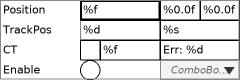
VISUALIZATION _VISU_WorkerDefGrid  // 240x80
VAR_IN_OUT
	m_Inst : FB_WorkerDefGrid;
END_VAR
    Rectangle (0,0 240x60)
    Rectangle (80,20 80x20), "%d", text variable: m_Inst._nTrackOffset
    Rectangle (0,0 80x20), "Position"
    Rectangle (0,20 80x20), "TrackPos"
    Rectangle (80,0 80x20), "%f", text variable: m_Inst.fPosition
        OnMouseClick: write the text variable via Default
    Rectangle (160,20 80x20), "%s", text variable: m_Inst._nTrackPosDomain
    Rectangle (160,0 40x20), "%0.0f", text variable: m_Inst._fPrintResolution
    Rectangle (200,0 40x20), "%0.0f", text variable: m_Inst._fSubPxResolution
    Rectangle (0,40 80x20), "CT"
    RoundedRectangle (80,40 20x20), colour toggle: m_Inst._pAttachedCt <> 0
    Rectangle (100,40 60x20), "%f", text variable: m_Inst.fCtPosition
    Rectangle (0,60 80x20), "Enable"
    Ellipse (80,60 20x20)
        toggle m_Inst.bWorkerEnable
    Rectangle (160,40 80x20), "Err: %d", text variable: m_Inst.nError, colour toggle: m_Inst.bError
    ComboBoxInteger (160,60 80x20), tooltip "LogLevel", variable: m_Inst._logLevel, text list: 'LogSeverity'
END_VISUALIZATION

(* stored: Version 1.1.0.1, ProductVersion 3.1.4024.11
   Visu _VISU_WorkerDefGrid: Id {6d8afdbb-2f0f-48ea-b77c-6f74e09f54ae} *)
